FUNCTION F_ConfigGroupEmulation




(********************************* Group *************************************
 Switching Group  
**********************************************************************************)
fbSG_001_Emulation.Config.Autostart := TRUE;


(********************************* Group *************************************
 Switching Group  
**********************************************************************************)
fbSG_002_Emulation.Config.Autostart := TRUE;

END_FUNCTION

(* stored: Version 1.1.0.1, ProductVersion 3.1.4024.9
   POU F_ConfigGroupEmulation: Id {c90ca705-efb5-4f58-829f-10c886e5e4eb}, SpecialFunc None *)
